// TIA Portal project "数字量，模拟量的学习" (V15.1)

(* hardware
DEVICE "S7-1200 station_1"  S7-1200 Station
   slot 0: "Rack_0"  S7-1200 Rack  Rack  V1.0
   slot 1: "PLC_1"  CPU 1214C DC/DC/Rly  6ES7 214-1HG40-0XB0  V4.2
*)

// ===== PLC "PLC_1"  CPU 1214C DC/DC/Rly =====

VAR_GLOBAL   // PLC tag table "默认变量表"
   "Tag_1" AT %MD200 : Real;
   "Tag_2" AT %MD204 : Real;
   "Tag_3" AT %MD208 : Real;
   "Tag_4" AT %MD2012 : Real;
   "Tag_5" AT %MW100 : Int;
   "Tag_6" AT %MW102 : Int;
   "Tag_7" AT %MD100 : DWord;
   "Tag_8" AT %MD104 : Real;
END_VAR

DATA_BLOCK "分数"   // DB1
{ S7_Optimized_Access := 'TRUE' }
VERSION : 0.1
   VAR
      考试分数 : Array[0..7] of Real;
   END_VAR
BEGIN
   考试分数[0] := 99.4;
   考试分数[1] := 100.0;
   考试分数[2] := 93.2;
   考试分数[3] := 80.5;
   考试分数[4] := 96.5;
   考试分数[5] := 96.1;
   考试分数[6] := 95.2;
   考试分数[7] := 98.0;
END_DATA_BLOCK

ORGANIZATION_BLOCK "Main"   // OB1, LAD, ProgramCycle
TITLE = "Main Program Sweep (Cycle)"
{ S7_Optimized_Access := 'TRUE' }
VERSION : 0.1
   VAR_INPUT
      Initial_Call : Bool;   // Initial call of this OB
      Remanence : Bool;   // =True, if remanent data are available
   END_VAR
BEGIN

REGION Network 1
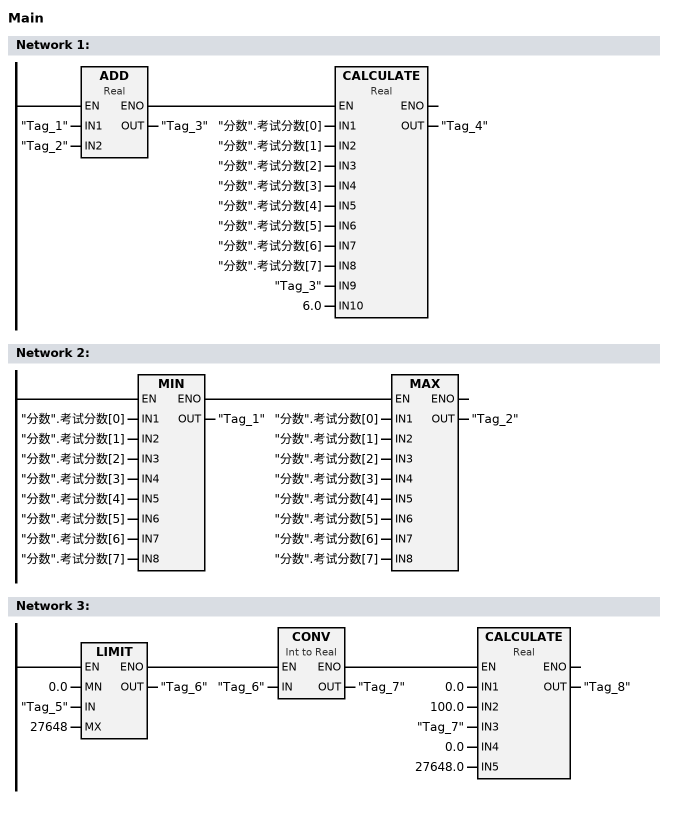
   RUNG wire#powerrail
      { S7_Templates := "SrcType := Real" } Add(in1 := "Tag_1", in2 := "Tag_2", out => "Tag_3")
      { S7_Templates := "SrcType := Real"; S7_Expression := "(IN1+IN2+IN3+IN4+IN5+IN6+IN7+IN8-IN9)/IN10" } Calculate(in1 := "分数".考试分数[0], in2 := "分数".考试分数[1], in3 := "分数".考试分数[2], in4 := "分数".考试分数[3], in5 := "分数".考试分数[4], in6 := "分数".考试分数[5], in7 := "分数".考试分数[6], in8 := "分数".考试分数[7], in9 := "Tag_3", in10 := 6.0, out => "Tag_4")
   END_RUNG
   // the same network as SCL:
   "Tag_3" := "Tag_1" + "Tag_2";
   "Tag_4" := ("分数".考试分数[0]+"分数".考试分数[1]+"分数".考试分数[2]+"分数".考试分数[3]+"分数".考试分数[4]+"分数".考试分数[5]+"分数".考试分数[6]+"分数".考试分数[7]-"Tag_3")/6.0;
END_REGION

REGION Network 2
   "Tag_1" := MIN(IN1 := "分数".考试分数[0], IN2 := "分数".考试分数[1], IN3 := "分数".考试分数[2], IN4 := "分数".考试分数[3], IN5 := "分数".考试分数[4], IN6 := "分数".考试分数[5], IN7 := "分数".考试分数[6], IN8 := "分数".考试分数[7]);
   "Tag_2" := MAX(IN1 := "分数".考试分数[0], IN2 := "分数".考试分数[1], IN3 := "分数".考试分数[2], IN4 := "分数".考试分数[3], IN5 := "分数".考试分数[4], IN6 := "分数".考试分数[5], IN7 := "分数".考试分数[6], IN8 := "分数".考试分数[7]);
END_REGION

REGION Network 3
   // no checked SCL form for this network; see the picture
END_REGION
END_ORGANIZATION_BLOCK